FUNCTION_BLOCK E_SWITCH (* Switching (demultiplexing) an event based on boolean input G *)
  (* Standard: 61499-1 Annex A; Description: Copyright (c) 2017 fortiss GmbH This program and the accompanying materials are made available under the terms of the Eclipse Public License 2.0 which is available at https://www.eclipse.org/legal/epl-2.0/ SPDX-License-Identifier: EPL-2.0 *)
  (* Version 1.0, 2017-09-21, Alois Zoitl, fortiss GmbH, initial API and implementation and/or initial documentation *)
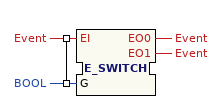
  EVENT_INPUT
    EI WITH G;
  END_EVENT
  EVENT_OUTPUT
    EO0;
    EO1;
  END_EVENT
  VAR_INPUT
    G : BOOL;
  END_VAR
END_FUNCTION_BLOCK
